{attribute 'pack_mode' := '1'}
TYPE ST_Disable EXTENDS ST_MsgToCCS:
STRUCT
END_STRUCT
END_TYPE

(* stored: Version 1.1.0.1, ProductVersion 3.1.4020.12
   DUT ST_Disable: Id {567212ce-5c5d-413f-abe9-b28a571d8615} *)
